Fanuc KAREL source: kx00013.KL

PROGRAM KX00013
%STACKSIZE=65535
%PRIORITY=65535
%NOLOCKGROUP
VAR
I : INTEGER
J : INTEGER
B : BOOLEAN
F : FILE
S : STRING[80]
P : XYZWPR
BEGIN
-- UNRESOLVED_PC line 11 opcodes [9C 4E] marker_code=0
END KX00013
